Staubli VAL3: check_solid.pjx

--- check_solid.pjx ---
Parameters version=s7.1 stackSize=5000 millimeterUnit=true
Program file=check_cube.pgx
Program file=check_cylinder.pgx
Program file=check_plane.pgx
Program file=check_sphere.pgx
Program file=create_cube.pgx
Program file=create_cylinder.pgx
Program file=create_easyCube.pgx
Program file=create_plane.pgx
Program file=create_sphere.pgx
Data file=check_solid.dtx

--- check_solid.dtx ---
mdesc mNomSpeed
bool bCreate_cube
bool bCreate_cylind
bool bCreate_plane
bool bCreate_sphere
frame fPlane = {fatherId=world[0]}
pointRx pOrigin_sphere = {fatherId=world[0]}
num nRadius_sphere
frame fCube = {fatherId=world[0]}
num nDistanceX_cube
num nDistanceY_cube
num nDistanceZ_cube
frame fCylinder = {fatherId=world[0]}
num nRadius_cyl
num nDistanceZ_cyl
pointRx pOrigin_cylind = {fatherId=world[0]}

--- check_cube.pgx ---
public program check_cube(tool x_tTool, bool& x_bCheck[])
  local point l_pPoint
  local bool l_bPositive
  local bool l_bNegative
begin
  //
  // CHECK IF THE TOOL IS INSIDE
  //
  x_bCheck=false
  //
  if bCreate_cube
    l_pPoint=here(x_tTool,fCube)
    // check if inside
    // x y z
    if l_pPoint.trsf.z>=-0.1 and l_pPoint.trsf.z<=nDistanceZ_cube
      // check if positive or negative of Y
      l_bPositive=l_pPoint.trsf.y>=-0.1 and l_pPoint.trsf.y<=nDistanceY_cube+0.1 and nDistanceY_cube>=-0.1
      l_bNegative=l_pPoint.trsf.y<=0.1 and l_pPoint.trsf.y>=nDistanceY_cube-0.1 and nDistanceY_cube<=0.1
      if l_bPositive or l_bNegative
        // check if positive or negative of X
        l_bPositive=l_pPoint.trsf.x>=-0.1 and l_pPoint.trsf.x<=nDistanceX_cube+0.1 and nDistanceX_cube>=-0.1
        l_bNegative=l_pPoint.trsf.x<=0.1 and l_pPoint.trsf.x>=nDistanceX_cube-0.1 and nDistanceX_cube<=0.1
        if l_bPositive or l_bNegative
          // is inside
          x_bCheck=true
        endIf
      endIf
    endIf
  endIf
end

--- check_cylinder.pgx ---
public program check_cylinder(tool x_tTool, bool& x_bCheck[])
  local point l_pPoint
  local point l_pNewOrigin
begin
  //
  // CHECK IF THE TOOL IS INSIDE
  //
  x_bCheck=false
  //
  if bCreate_cylind
    l_pPoint=here(x_tTool,fCube)
    // check if inside
    if l_pPoint.trsf.z>=-0.1 and l_pPoint.trsf.z<=nDistanceZ_cyl
      // inside the cylinder
      l_pNewOrigin=compose(pOrigin_cylind,world,{0,0,l_pPoint.trsf.z,0,0,0})
      if distance(l_pNewOrigin,l_pPoint)<=nRadius_cyl
        // is inside
        x_bCheck=true
      endIf
    endIf
  endIf
end

--- check_plane.pgx ---
public program check_plane(tool x_tTool, bool& x_bCheck[])
  local point l_pPoint
begin
  //
  // CHECK IF THE TOOL IS INSIDE
  //
  x_bCheck=false
  //
  if bCreate_plane
    l_pPoint=here(x_tTool,fPlane)
    // check if inside
    if l_pPoint.trsf.z<=0.1
      // set to TRUE
      x_bCheck=true
    endIf
  endIf
end

--- check_sphere.pgx ---
public program check_sphere(tool x_tTool, bool& x_bCheck[])
  local point l_pPoint
begin
  //
  // CHECK IF THE TOOL IS INSIDE
  //
  x_bCheck=false
  //
  if bCreate_sphere
    l_pPoint=here(x_tTool,world)
    // sphere
    if distance(pOrigin_sphere,l_pPoint)<=nRadius_sphere
      // check if inside
      x_bCheck=true
    endIf
  endIf
end

--- create_cube.pgx ---
public program create_cube(point x_pOrigin, point x_pPointX, point x_pPointY, num x_nDistanceZ)
  local trsf l_trsfCopy
  local point l_pPoint
begin
  //
  // build the cube
  // Origin
  if setFrame(x_pOrigin,x_pPointX,x_pPointY,fCube)==0
    bCreate_cube=true
  endIf
  // Distance x y z
  // X AXES
  l_pPoint.trsf=position(x_pPointX,fCube)
  nDistanceX_cube=l_pPoint.trsf.x
  // Y AXES
  l_pPoint.trsf=position(x_pPointY,fCube)
  nDistanceY_cube=l_pPoint.trsf.y
  // Z distance
  nDistanceZ_cube=x_nDistanceZ
end

--- create_cylinder.pgx ---
public program create_cylinder(point x_pOrigin, num x_nRadius, num x_nDistanceZ)
begin
  //
  // build the Cylinder
  //
  if setFrame(x_pOrigin,compose(x_pOrigin,world,{x_nRadius,0,0,0,0,0}),compose(x_pOrigin,world,{0,x_nRadius,0,0,0,0}),fCylinder)==0
    bCreate_cylind=true
  else
    bCreate_cylind=false
  endIf
  // copy all
  nRadius_cyl=x_nRadius
  nDistanceZ_cyl=x_nDistanceZ
  pOrigin_cylind.trsf=position(x_pOrigin,world)
end

--- create_easyCube.pgx ---
public program create_easyCube(point x_pOrigin, num x_nDistanceX, num x_nDistanceY, num x_nDistanceZ)
  local trsf l_trsfCopy
begin
  //
  // build the cube
  // Origin
  if setFrame(x_pOrigin,compose(x_pOrigin,world,{x_nDistanceX,0,0,0,0,0}),compose(x_pOrigin,world,{0,x_nDistanceY,0,0,0,0}),fCube)==0
    bCreate_cube=true
  else
    bCreate_cube=false
  endIf
  // Distance x y z
  nDistanceX_cube=x_nDistanceX
  nDistanceY_cube=x_nDistanceY
  nDistanceZ_cube=x_nDistanceZ
  // regolate the frame
  l_trsfCopy=fCube.trsf
  fCube.trsf={l_trsfCopy.x,l_trsfCopy.y,l_trsfCopy.z,0,0,0}
end

--- create_plane.pgx ---
public program create_plane(point x_pOrigin, point x_pPointX, point x_pPointY)
begin
  //
  // build the plane
  //
  // Origin
  if setFrame(x_pOrigin,x_pPointX,x_pPointY,fPlane)==0
    bCreate_plane=true
  else
    bCreate_plane=false
  endIf
end

--- create_sphere.pgx ---
public program create_sphere(point x_pOrigin, num x_nRadius)
begin
  //
  // build the sphere
  //
  // Origin
  pOrigin_sphere.trsf=position(x_pOrigin,world)
  bCreate_sphere=true
  // Radius
  nRadius_sphere=x_nRadius
end
